FUNCTION_BLOCK ABSTRACT ChamberBase EXTENDS TExecution IMPLEMENTS IDevice
VAR_INPUT
	IoChamberBase : IoChamberBase;
END_VAR
VAR_OUTPUT
END_VAR
VAR
	{attribute 'OPC.UA.DA' := '0'}
	_name : STRING;
	{attribute 'OPC.UA.DA' := '0'}
	_deviceID : STRING;				
	{attribute 'OPC.UA.DA' := '0'}
	_family : DeviceFamily := DeviceFamily.Chamber;		
	{attribute 'OPC.UA.DA' := '0'}
	_logger : Logger;
	{attribute 'OPC.UA.DA' := '0'}
	_message : StringBuilder;
	{attribute 'OPC.UA.DA' := '0'}
	_chamberConfig : DeviceConfiguration;
	
	{attribute 'OPC.UA.DA' := '0'}
	InputIsInMaintenanceMode AT %I* : BOOL;
	{attribute 'OPC.UA.DA' := '0'}
	InputIsInRunMode AT %I* : BOOL;
	{attribute 'OPC.UA.DA' := '0'}
	InputArmNotExtended	AT %I* : BOOL;		
	
	{attribute 'OPC.UA.DA' := '0'}
	_lifeTimeCount : UINT;
	{attribute 'OPC.UA.DA' := '0'}
	_notifyIsAlive : BOOL;
	{attribute 'OPC.UA.DA' := '0'}
	_pulseIsAliveGenerator : TON;
	{attribute 'OPC.UA.DA' := '0'}
	_pulseGeneratorBase : TON;
	{attribute 'OPC.UA.DA' := '0'}
	_execPulseGeneratorBase : TON;	
	
	{attribute 'OPC.UA.DA' := '0'}
	_itemSchedulerBase : INT;
	{attribute 'OPC.UA.DA' := '0'}
	_itemExecSchedulerBase : INT;
	{attribute 'OPC.UA.DA' := '0'}
	_itemRaisedPropertiesBase : INT;	
	
	{attribute 'OPC.UA.DA' := '0'}
	_deliverMessagesBase : INT;
		
	{attribute 'OPC.UA.DA' := '0'}
	_armNotExtendedCmd : BOOL;	
	{attribute 'OPC.UA.DA' := '0'}			  		   
	_raisePropertiesBase : BOOL;	 
	
	{attribute 'OPC.UA.DA' := '0'}
	_extendsArm : BOOL;
	
	StateMsg : STRING(255);
	IsAliveMsg : STRING(255);
	IsInMaintenanceMsg : STRING(255);
	ArmNotExtendedMsg : STRING(255);
	EfemSlitDoorOpenPositionMsg : STRING(255);
	IsReadyToLoadUnloadMsg : STRING(255);	

	{attribute 'OPC.UA.DA' := '0'}
	_slitDoorPosition : ESlitDoorPosition;
	{attribute 'OPC.UA.DA' := '0'}
	_slitDoorOpenPosition : BOOL;
	{attribute 'OPC.UA.DA' := '0'}
	_slitDoorClosePosition : BOOL;
	
	{attribute 'OPC.UA.DA' := '0'}
	ioMessage : STRING;
	
	{attribute 'OPC.UA.DA' := '0'}
	_stageIsInLoadingPosition : BOOL;
END_VAR

// Check if it's still alive	
IF _notifyIsAlive THEN
	IsAliveMsg := TO_STRING(_lifeTimeCount);
	_notifyIsAlive := FALSE;
END_IF

IF HardwareGlobalVariables.ChamberState <> State THEN
	HardwareGlobalVariables.ChamberState := State;
	StateMsg := ANY_TO_STRING(State);		
END_IF


CASE _deliverMessagesBase OF		
	EFeedbackMsgChamberBase.IsInMaintenanceMsg :		
		IsInMaintenanceMsg := ioMessage;	
			
	EFeedbackMsgChamberBase.ArmNotExtendedMsg :				
		ArmNotExtendedMsg := ioMessage;	

	EFeedbackMsgChamberBase.EfemSlitDoorOpenPositionMsg :		
		EfemSlitDoorOpenPositionMsg := ioMessage;	
			
	EFeedbackMsgChamberBase.IsReadyToLoadUnloadMsg :				
		IsReadyToLoadUnloadMsg := ioMessage;	
		
END_CASE

RaisePropertiesChangedBase(_raisePropertiesBase);

IF NOT _armNotExtendedCmd AND NOT _raisePropertiesBase THEN
	MessageSchedulerBase();	
END_IF

{attribute 'TcRpcEnable' := '1'}
METHOD PROTECTED ArmExtendEnabled 
VAR_INPUT
	Execute : BOOL;
	ExtendsArm : BOOL;
END_VAR
VAR
END_VAR
IF Execute THEN	
	(*_armNotExtendedCmd := TRUE;	
	
	_extendsArm := ExtendsArm;

	IF _execPulseGeneratorBase.Q THEN
		_execPulseGeneratorBase(IN := FALSE, PT := T#10MS);
			
		CASE _itemExecSchedulerBase OF
			0:  OutputArmExtendEnabled := _extendsArm;
			
				_logger.Information(_message.Reset().Append('ArmExtendEnabled : ').Append(TO_STRING(_extendsArm)).ToString());			   					
				_itemExecSchedulerBase := 1;
			
			1:  _armNotExtendedCmd := FALSE;	
				_itemExecSchedulerBase := 0;		
								
		END_CASE
	ELSE
		_execPulseGeneratorBase(IN := TRUE, PT := T#50MS);	
	END_IF*)
END_IF
END_METHOD

PROPERTY DeviceID : STRING
GET
DeviceID := _deviceID;
END_GET
SET
_deviceID := DeviceID;
END_SET
END_PROPERTY

PROPERTY Family : DeviceFamily
GET
Family := _family;
END_GET
SET
_family := Family;
END_SET
END_PROPERTY

METHOD GetArmNotExtended
VAR_INPUT
END_VAR
_deliverMessagesBase := EFeedbackMsgChamberBase.ArmNotExtendedMsg;
ioMessage := ANY_TO_STRING(NOT InputArmNotExtended);
END_METHOD

METHOD PROTECTED IsAlive
VAR_INPUT
END_VAR
_notifyIsAlive := TRUE;

IF _lifeTimeCount < 5 THEN
	_lifeTimeCount := _lifeTimeCount + 1;
ELSE
	_lifeTimeCount := 1;
END_IF
END_METHOD

METHOD IsInMaintenance 
VAR_INPUT
END_VAR
_deliverMessagesBase := EFeedbackMsgChamberBase.IsInMaintenanceMsg;

IF InputIsInMaintenanceMode AND NOT InputIsInRunMode THEN
	ioMessage := TO_STRING(TRUE);
ELSIF InputIsInMaintenanceMode AND InputIsInRunMode THEN
ioMessage := TO_STRING(FALSE);
ELSE
	ioMessage := TO_STRING(FALSE);
END_IF
END_METHOD

METHOD IsReadyToLoadUnload
VAR_INPUT
END_VAR
_deliverMessagesBase := EFeedbackMsgChamberBase.IsReadyToLoadUnloadMsg;

// Conditions for authorising the arm to enter the chamber
IF IoChamberBase.InputEfemSlitDoorOpen AND StageIsInLoadingPosition THEN	
	IoChamberBase.OutputIsReadyToLoadUnload := TRUE;
ELSE
	IoChamberBase.OutputIsReadyToLoadUnload := FALSE;
END_IF

ioMessage := ANY_TO_STRING(IoChamberBase.OutputIsReadyToLoadUnload);
END_METHOD

METHOD MessageSchedulerBase
VAR_INPUT
END_VAR
IF _pulseGeneratorBase.Q THEN
	_pulseGeneratorBase(IN := FALSE, PT := T#10MS);
		
	CASE _itemSchedulerBase OF			
		0:  _deliverMessagesBase := EFeedbackMsgChamberBase.IsInMaintenanceMsg;
			ioMessage := ' ';
			_itemSchedulerBase := 1;
			
		1:	IsInMaintenance(); 
			_itemSchedulerBase := 2;

		2:  _deliverMessagesBase := EFeedbackMsgChamberBase.ArmNotExtendedMsg;
			ioMessage := ' ';
			_itemSchedulerBase := 3;
			
		3:	GetArmNotExtended(); 
			_itemSchedulerBase := 4;	
			
		4:  _deliverMessagesBase := EFeedbackMsgChamberBase.EfemSlitDoorOpenPositionMsg; 
			ioMessage := ' ';		
			_itemSchedulerBase := 5;
			
		5:	ReadEfemSlitDoorPosition(); 
			_itemSchedulerBase := 6;	
			
		6:	_deliverMessagesBase := EFeedbackMsgChamberBase.IsReadyToLoadUnloadMsg;
			ioMessage := ' ';
		   _itemSchedulerBase := 7;
		   
		7:	IsReadyToLoadUnload(); 
			_itemSchedulerBase := 0;	
		
	END_CASE
ELSE
	_pulseGeneratorBase(IN := TRUE, PT := T#50MS);		
END_IF


IF _pulseIsAliveGenerator.Q THEN
	_pulseIsAliveGenerator(IN := FALSE, PT := T#10MS);
		
	IsAlive();	
ELSE
	_pulseIsAliveGenerator(IN := TRUE, PT := T#1000MS);		
END_IF
END_METHOD

{attribute 'TcRpcEnable' := '1'}
METHOD ABSTRACT MoveSlitDoorPosition
VAR_INPUT
	Execute : BOOL;
	Position : INT;
END_VAR
END_METHOD

PROPERTY Name : STRING
GET
Name := _name;
END_GET
SET
_name := Name;
END_SET
END_PROPERTY

{attribute 'TcRpcEnable' := '1'}
METHOD RaisePropertiesChangedBase
VAR_INPUT
	Execute : BOOL;
END_VAR
IF Execute THEN		
	_raisePropertiesBase := TRUE;	
	
	IF _pulseGeneratorBase.Q THEN
		_pulseGeneratorBase(IN := FALSE, PT := T#10MS);
		
		CASE _itemRaisedPropertiesBase OF		
			0: IsInMaintenanceMsg := ' ';
				_itemRaisedPropertiesBase := 1;
			
			1: ArmNotExtendedMsg := ' ';		   
				_itemRaisedPropertiesBase := 10;
				
			10: 
				_logger.Information(_message.Reset().
								    Append(_chamberConfig.Name).
								    Append(' - RaisePropertiesChangedBase').ToString());
				_raisePropertiesBase := FALSE;
				_itemRaisedPropertiesBase := 0;
		
		END_CASE
	
	ELSE
		_pulseGeneratorBase(IN := TRUE, PT := T#50MS);	
	END_IF
		
END_IF
END_METHOD

METHOD ReadEfemSlitDoorPosition
VAR_INPUT
END_VAR
_deliverMessagesBase := EFeedbackMsgChamberBase.EfemSlitDoorOpenPositionMsg;

ioMessage := ANY_TO_STRING(IoChamberBase.InputEfemSlitDoorOpen);
END_METHOD

METHOD ABSTRACT ReadSlitDoorPosition
VAR_INPUT
END_VAR
END_METHOD

PROPERTY PUBLIC SlitDoorClosePosition : BOOL
GET
SlitDoorClosePosition := _slitDoorClosePosition;
END_GET
SET
_slitDoorClosePosition := SlitDoorClosePosition;
END_SET
END_PROPERTY

PROPERTY PUBLIC SlitDoorOpenPosition : BOOL
GET
SlitDoorOpenPosition := _slitDoorOpenPosition;
END_GET
SET
_slitDoorOpenPosition := SlitDoorOpenPosition;
END_SET
END_PROPERTY

PROPERTY PUBLIC SlitDoorPosition : ESlitDoorPosition
GET
SlitDoorPosition := _slitDoorPosition;
END_GET
SET
_slitDoorPosition := SlitDoorPosition;
END_SET
END_PROPERTY

PROPERTY PUBLIC StageIsInLoadingPosition : bool
GET
StageIsInLoadingPosition := _stageIsInLoadingPosition;
END_GET
SET
_stageIsInLoadingPosition := StageIsInLoadingPosition;
END_SET
END_PROPERTY

END_FUNCTION_BLOCK

(* stored: Version 1.1.0.1, ProductVersion 3.1.4024.12
   POU ChamberBase: Id {fb75d943-5c54-4f31-871f-76b380309cb1}, SpecialFunc None
   Folder Commands: Id {87dbbb78-d556-4bee-9f17-98438344acd5}
   Method ArmExtendEnabled: Id {527959d9-7c3e-4f1b-a463-15fbb46976ea}
   Property DeviceID: Id {00424e6b-0a76-40f0-a94a-76a014c72092}
   Get Get: Id {22831275-1cce-4662-b96f-09e9a2427fee}
   Set Set: Id {5e0d27fd-e715-48c3-964f-6adcd311c3fa}
   Property Family: Id {638f86d8-8e91-4299-a80b-5f082a0532b4}
   Get Get: Id {fc70de96-6c14-49c9-82d1-69b7019e858e}
   Set Set: Id {abb4cf80-0a3a-4a3a-be06-43e676907630}
   Method GetArmNotExtended: Id {267eb2b5-fbe1-436b-8d75-0c88f9cfc35f}
   Method IsAlive: Id {e672f27a-afc0-43a6-863b-abe4dc0b496d}
   Method IsInMaintenance: Id {b36b95b2-6900-47ee-b8a2-310a4b643a5d}
   Method IsReadyToLoadUnload: Id {9119baf5-8db6-4866-8457-a413aa4fb030}
   Method MessageSchedulerBase: Id {5a6545ee-559c-4456-ac8d-8b6269c847ed}
   Method MoveSlitDoorPosition: Id {ee0dafd3-440f-43c1-85f1-91448019e241}
   Property Name: Id {f0414c56-d676-4440-b6cc-8e0550ec35a4}
   Get Get: Id {a4b151ec-ebb5-4bca-bad5-38b703610f76}
   Set Set: Id {020571c0-1270-4f7b-84ee-f41cf3c87513}
   Method RaisePropertiesChangedBase: Id {8268f1b3-d357-4a2e-a702-a6e496723a17}
   Method ReadEfemSlitDoorPosition: Id {86634d83-e723-4261-89f2-6fff79ac95d0}
   Method ReadSlitDoorPosition: Id {aea0058d-e4a6-4853-8d42-b50dbb531c7d}
   Property SlitDoorClosePosition: Id {4979245c-5e35-45bc-a877-f4c7c89f9513}
   Get Get: Id {6382749c-9f87-4008-a645-c60d466bf462}
   Set Set: Id {eaf6d173-7aa2-4025-99c2-56eea569524c}
   Property SlitDoorOpenPosition: Id {fd8a629d-4672-4f0f-b941-baf4260892d8}
   Get Get: Id {47c1b292-545c-4ad2-92bc-ca6c7dc7b5b6}
   Set Set: Id {d4e67467-3076-4b9f-aecd-86c2e174ded1}
   Property SlitDoorPosition: Id {8852f7f4-18df-4547-8f8e-31cc39cd4fb5}
   Get Get: Id {229f2151-13aa-4f0a-a694-8277d758a5ce}
   Set Set: Id {3711938b-1f0d-4fea-9852-b428991e0861}
   Property StageIsInLoadingPosition: Id {0c875471-5161-43d0-8184-2f8d9347d8d4}
   Get Get: Id {4c0e5e2c-cb8d-4eba-a3c9-a3ec32fa92b4}
   Set Set: Id {aafdccf8-691a-4d71-9e38-446a9d7f1403} *)
